(* PLC project Tc2_Utilities.STRING_TO_GUID Demo, tc3-libraries-kb TwinCAT 3.1 *)
(* stored: creationDateTime 2026-05-10T19:00:00, modificationDateTime 2026-05-10T19:00:00 *)

PROGRAM P_Demo_STRING_TO_GUID
  VAR
    rResult : GUID;  (* STRING_TO_GUID 返回值 *)
    bRun : BOOL;  (* 触发一次调用 *)
    s : STRING := '12345678-1234-1234-1234-123456789ABC';  (* 测试用本地变量 *)
  END_VAR

            // ============================================================
// Tc2_Utilities.STRING_TO_GUID 演示程序（FUNCTION）
// ============================================================
// 验证步骤：
//   1. 引用 Tc2_Utilities
//   2. 编译 + 登录
//   3. 强制 bRun := TRUE 一个周期
//   4. 在线监视 rResult / 各 demo 变量
// ============================================================

IF bRun THEN
    rResult := STRING_TO_GUID(s);
    bRun := FALSE;
END_IF;

          
END_PROGRAM
